FUNCTION_BLOCK TcCommand IMPLEMENTS itfCommand
//VAR_INPUT
//END_VAR
//VAR_OUTPUT
//END_VAR
VAR
	_Command        : ST_Command;	
END_VAR

{warning 'add method implementation '}
METHOD Abort : MC_Error
VAR
	
END_VAR
END_METHOD

{warning 'add property implementation'}
PROPERTY Active : BOOL
GET
Active := _Command.Active;
END_GET
SET
_Command.Active := Active;
END_SET
END_PROPERTY

{warning 'add property implementation'}
PROPERTY Busy : BOOL
GET
Busy := _Command.Busy;
END_GET
SET
_Command.Busy := Busy;
END_SET
END_PROPERTY

{warning 'add property implementation'}
PROPERTY Command : MC_COMMAND_REF
GET
Command := _Command.Command;
END_GET
SET
 _Command.Command :=  Command;
END_SET
END_PROPERTY

{warning 'add property implementation'}
PROPERTY CommandAborted : BOOL
GET
CommandAborted := _Command.CommandAborted;
END_GET
SET
 _Command.CommandAborted := CommandAborted;
END_SET
END_PROPERTY

{warning 'add property implementation'}
PROPERTY Done : BOOL
GET
Done := _Command.Done;
END_GET
SET
_Command.Done := Done;
END_SET
END_PROPERTY

{warning 'add property implementation'}
PROPERTY Error : BOOL
GET
Error := _Command.Error;
END_GET
SET
_Command.Error := Error;
END_SET
END_PROPERTY

{warning 'add property implementation'}
PROPERTY ErrorId : MC_Error
GET
ErrorId := _Command.ErrorId;
END_GET
SET
_Command.ErrorId := ErrorId;
END_SET
END_PROPERTY

PROPERTY ErrorID_Udint : UDINT
GET
ErrorID_Udint := _Command.ErrorID_Udint;
END_GET
SET
_Command.ErrorID_Udint := ErrorID_Udint;
END_SET
END_PROPERTY

PROPERTY Status : BOOL
GET
Status :=  _Command.Status;
END_GET
SET
 _Command.Status := Status;
END_SET
END_PROPERTY

{warning 'add method implementation '}
METHOD Wait : MC_Error (* This method only makes sense in the IEC 61499 environment*)
VAR_INPUT
	Timeout	: TIME;
	AbortOnTimeout	: BOOL;
END_VAR
VAR
	
END_VAR
END_METHOD

END_FUNCTION_BLOCK

(* stored: Version 1.1.0.1, ProductVersion 3.1.4024.12
   POU TcCommand: Id {b41e1980-0cf0-4034-bd15-e55e20969f1a}, SpecialFunc None
   Method Abort: Id {a0de7d3b-923f-4416-b4ef-58c6f46dbf33}
   Property Active: Id {fd3da06e-f2a5-45d4-8e0d-ca1c7b52e98a}
   Get Get: Id {fc3a9126-fa71-4806-b52e-5be02e326a45}
   Set Set: Id {d3b187d2-c717-4608-970a-ecf94d5b6d29}
   Property Busy: Id {c70f78a5-d31f-4558-8325-7a017493ec48}
   Get Get: Id {ad9f33f6-5e4a-45f0-9497-56006533bd89}
   Set Set: Id {18549f46-ae12-4851-b3b6-82358cd2d53a}
   Property Command: Id {1e98e78f-e26d-4d3f-9df5-62d3db7c2351}
   Get Get: Id {e45bb2ab-5252-4ad9-a904-38438153e8c7}
   Set Set: Id {8c572b14-e4a4-4892-92bc-7bfb6fccf1a4}
   Property CommandAborted: Id {64fc8e8b-1fca-4237-b95d-a22ade7daee5}
   Get Get: Id {c7567f4a-3327-41fc-9556-98ccbf68eaa5}
   Set Set: Id {fa72ceb7-81cf-4104-8e08-990f919ec723}
   Property Done: Id {612a916d-4670-4f93-a6db-9618fe011e35}
   Get Get: Id {90c3e97a-8375-42bb-8d60-3a9a9157b587}
   Set Set: Id {27a7b96b-ffe3-40bd-b916-c07758186070}
   Property Error: Id {1a6ee7c5-9948-479d-8097-45d267cf7820}
   Get Get: Id {633f7a6f-d36e-45e7-b168-a50576d4d3d1}
   Set Set: Id {0ee27777-a1a1-4c3c-9011-4eafcc1a9553}
   Property ErrorId: Id {695df361-2c8d-4b04-9259-0517f9e43c3e}
   Get Get: Id {fd1cbed5-a888-4458-8c8c-689361eb11e5}
   Set Set: Id {bfdfeb48-a86d-40e7-88a0-17dcfbbe14f3}
   Property ErrorID_Udint: Id {0b4a8509-d39f-448d-9a5c-d564f1c9dff4}
   Get Get: Id {aadc048e-1c35-429c-ba68-27b3e12591ea}
   Set Set: Id {28310b40-fca3-4bf7-8f8e-249432b561d6}
   Property Status: Id {e87e1294-d370-4e44-93c9-63423bcbc013}
   Get Get: Id {2aba010c-9b62-4358-824a-10dcc9453fd3}
   Set Set: Id {8a415b82-65e1-419b-a1bc-7dd5d1d14034}
   Method Wait: Id {265638f0-0d66-4716-91e3-9998c65eddaf} *)
